(* IEC 61131-3 sources: 89152_FlorisHendrix_AfstudeerProject/89152_FlorisHendrix_ExamenProject/Stations/Terminal/HMI/Class/_Lse (part 3) *)

END_FUNCTION

FUNCTION VIRTUAL GLOBAL _Lse::SCROLL_GetLinePosition
VAR_INPUT
  pt1 : ^_SCROLL;
  y   : UINT;
  pr  :^_ROOM;
END_VAR

  GetLinePosition_SCROLL(pt1, y, pr);

END_FUNCTION

FUNCTION VIRTUAL GLOBAL _Lse::SCROLL_OutLine
VAR_INPUT
  pt1   : ^_SCROLL;
  y     : UINT;
  no    : UINT;
  beam  : BOOL;
END_VAR

  OutLine_SCROLL(pt1, y, no, beam, TRUE);

END_FUNCTION

FUNCTION VIRTUAL GLOBAL _Lse::SCROLL_Beam
VAR_INPUT
  pt1   : ^_SCROLL;
  y     : UINT;
  no    : UINT;
  state : BOOL;
END_VAR

  Beam_SCROLL(pt1, y, no, state);

END_FUNCTION

FUNCTION VIRTUAL GLOBAL _Lse::SCROLL_ActBeam
VAR_INPUT
  pt1   : ^_SCROLL;
  state : BOOL;
END_VAR

  ActBeam_SCROLL(pt1, state);

END_FUNCTION

FUNCTION VIRTUAL GLOBAL _Lse::SCROLL_Draw
VAR_INPUT
  pt1  : ^_SCROLL;
  beam : BOOL;
END_VAR

  Draw_SCROLL(pt1, beam);

END_FUNCTION

FUNCTION VIRTUAL GLOBAL _Lse::SCROLL_Start
VAR_INPUT
  pt1 : ^_SCROLL;
END_VAR

  Start_SCROLL(pt1, TRUE);

END_FUNCTION

FUNCTION VIRTUAL GLOBAL _Lse::SCROLL_Ready
VAR_INPUT
  pt1  : ^_SCROLL;
  beam : BOOL;
END_VAR

  Ready_SCROLL(pt1, beam);

END_FUNCTION

FUNCTION VIRTUAL GLOBAL _Lse::SCROLL_Run
VAR_INPUT
  pt1    : ^_SCROLL;
  pevent : ^_EVENT;
END_VAR

  Run_SCROLL(pt1, pevent);

END_FUNCTION

FUNCTION VIRTUAL GLOBAL _Lse::SCROLL_End
VAR_INPUT
  pt1 : ^_SCROLL;
END_VAR

  End_SCROLL(pt1);

END_FUNCTION

FUNCTION VIRTUAL GLOBAL _Lse::SCROLL_OutPage
VAR_INPUT
  pt1 : ^_SCROLL;
END_VAR

  OutPage_SCROLL(pt1);

END_FUNCTION

FUNCTION VIRTUAL GLOBAL _Lse::SCROLL_ScrollUp
VAR_INPUT
  pt1 : ^_SCROLL;
END_VAR

  ScrollUp_SCROLL(pt1);

END_FUNCTION

FUNCTION VIRTUAL GLOBAL _Lse::SCROLL_ScrollDown
VAR_INPUT
  pt1 : ^_SCROLL;
END_VAR

  ScrollDown_SCROLL(pt1);

END_FUNCTION

FUNCTION VIRTUAL GLOBAL _Lse::SCROLL_GetPosition
VAR_INPUT
  pt1 : ^_SCROLL;
END_VAR
VAR_OUTPUT
  retcode : UINT;
END_VAR

  retcode := GetPosition_SCROLL(pt1);

END_FUNCTION

FUNCTION VIRTUAL GLOBAL _Lse::SCROLL_level_draw
VAR_INPUT
  pt1   : ^_LEVEL;
  horiz : BOOL;
END_VAR

  level_draw(pt1, horiz, TRUE);

END_FUNCTION

FUNCTION VIRTUAL GLOBAL _Lse::SCROLL_level_run
VAR_INPUT
  pt1   : ^_LEVEL;
  no    : DINT;
  pos   : DINT;
  horiz : BOOL;
END_VAR

  level_run(pt1, no, pos, horiz);

END_FUNCTION

FUNCTION __CDECL VIRTUAL GLOBAL _Lse::IF_SoftReset

  DownloadState := 2;

END_FUNCTION

FUNCTION __CDECL VIRTUAL GLOBAL _Lse::IF_UserStation
	VAR_INPUT
		station 	: UINT;
		pcd 	: ^_COMDEF;
		pobserve 	: ^BOOL;
	END_VAR
	VAR_OUTPUT
		retcode 	: BOOL;
	END_VAR
  VAR
	  no   : UDINT;
    ppp  : ^_POINTERPARA;
  END_VAR

  retcode    := true;
  no  := UserGlobal.no;
  ppp := UserGlobal.ptr;
  while no do
    no  -= 1;
    if(ppp^.ptr$^_Global^.IF_UserStation(station, pcd, pobserve) = false) then
      retcode := false;
    end_if;
    ppp += sizeof(_POINTERPARA);
  end_while;

END_FUNCTION

FUNCTION __CDECL VIRTUAL GLOBAL _Lse::IF_CantWriteNoAccess
	VAR_INPUT
		pres 	: ^_RESULT;
		pvl 	: ^_VARLABEL;
	END_VAR
	VAR_OUTPUT
		retcode 	: BOOL;
	END_VAR
  VAR
	  no   : UDINT;
    ppp  : ^_POINTERPARA;
  END_VAR

  retcode := false;
  no  := UserGlobal.no;
  ppp := UserGlobal.ptr;
  while no do
    no  -= 1;
    if(ppp^.ptr$^_Global^.IF_CantWriteNoAccess(pres, pvl) = true) then
      retcode := true;
    end_if;
    ppp += sizeof(_POINTERPARA);
  end_while;

END_FUNCTION

FUNCTION VIRTUAL GLOBAL _Lse::ActivateBubbleHelp::Write
	VAR_INPUT
		input (EAX) 	: DINT;
	END_VAR
	VAR_OUTPUT
		result (EAX) 	: DINT;
	END_VAR

	ActivateBubbleHelp := input;
 	result := ActivateBubbleHelp;

  if(result <> 0) then
    InsertCmd(CMD_KILLEDITOR, 0, 0);
  end_if;

END_FUNCTION

FUNCTION __CDECL GLOBAL Thread2_AddCmd
  VAR_INPUT
    pcmd : ^_Thread2CmdLine;
  END_VAR
  VAR_OUTPUT
    retcode : bool;
  END_VAR

  retcode := false;

  if(pcmd^.cmd <> T2_NONE) then
    if(MailBox2Handle <> NIL) then
      if(OS_MT_PutCond(MailBox2Handle, pcmd) = 1) then
        retcode := true;
      end_if;
    end_if;
  end_if;

END_FUNCTION

FUNCTION __CDECL GLOBAL _Lse::Thread2
	VAR_INPUT
		pthis 	: ^void;
	END_VAR
  VAR
  	t2cmdline : _Thread2CmdLine;
  END_VAR

  this := pthis$^_Lse;

  while(1) do
    if(OS_MT_GET(MailBox2Handle, #t2cmdline) = MTERROR_NONE) then // wait for cmd in mailbox
      RTK_Thread2(#t2cmdline);
    end_if;
    OS_MT_DELAY(1);
  end_while;

END_FUNCTION

FUNCTION __CDECL VIRTUAL GLOBAL _Lse::IF_WindowMoveable
	VAR_INPUT
		whoami 	: ^_WHOAMI;
	END_VAR
	VAR_OUTPUT
		retcode 	: BOOL;
	END_VAR
  VAR
    pp  : ^_PICPOI;
	  no  : UDINT;
    ppp : ^_POINTERPARA;
  END_VAR

  retcode := true;

  if(GlobalBitState and GLOBAL_BIT_IFWINMOVEABLE) then
    no  := UserGlobal.no;
    ppp := UserGlobal.ptr;
    while no do
      if(ppp^.para and GLOBAL_BIT_IFWINMOVEABLE) then
        if(ppp^.ptr$^_Global^.IF_WindowMoveable(whoami) = false) then
          retcode := false;
          return;
        end_if;
      end_if;
	    no  -= 1;
	    ppp += sizeof(_POINTERPARA);
    end_while;
  end_if;

  pp := FindScreen(whoami);
  if(pp <> NIL) then
    if(pp^.ptr$^_Screen^.S_WindowMoveable() = false) then
      retcode := false;
    end_if;
  end_if;

END_FUNCTION

FUNCTION __CDECL VIRTUAL GLOBAL _Lse::IF_Progress
	VAR_INPUT
		pscan 	: ^_SCAN;
		visible 	: BOOL;
	END_VAR
  VAR
	  no  : UDINT;
    ppp : ^_POINTERPARA;
  END_VAR

  no  := UserGlobal.no;
  ppp := UserGlobal.ptr;
  while no do
    ppp^.ptr$^_Global^.IF_Progress(pscan, visible);
    no  -= 1;
    ppp += sizeof(_POINTERPARA);
  end_while;

END_FUNCTION
